// Mitsubishi GX Works2 project: 28-05-2020 SFC   PLC: FX3U/FX3UC

PROGRAM MAIN
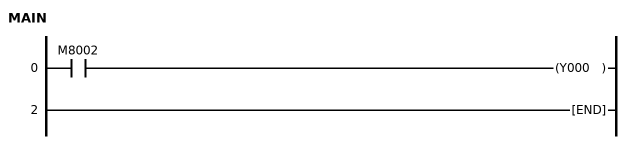
0     LD      M8002
      OUT     Y000
2     END
END_PROGRAM
